   tongsocot = SmartTags("Blister_Show_Total_Blister_Column")	
   'tongsocot = 6
   '-------------------
   'bung = tongsocot - 1
   'If bung < 1 Then
   'bung = 1
   'End If
   '-------------------
   cycle = kc_hieudung / tongsocot '137
   Do_rong_cot = (cycle/3) *2		'91,3
   
   kc_2_cot = cycle		
   
   cot = tongsocot
   
   If tongsocot > 1 Then
   letrai = 50	
   Blis(tongsocot).width =  Do_rong_cot 
   	
   For i = 2  To tongsocot
   cot = cot - 1
   letrai = letrai + kc_2_cot
   
   Blis(cot).left =  letrai 
   Blis(cot).width = Do_rong_cot
   Next
   
   End If

VB script "Check_Lot"
   'Tip:
   ' 1. Use the <CTRL+SPACE> or <CTRL+I> shortcut to open a list of all objects and functions
   ' 2. Write the code using the HMI Runtime object.
   '  Example: HmiRuntime.Screens("Screen_1").
   ' 3. Use the <CTRL+J> shortcut to create an object reference.
   'Write the code as of this position:
   
   If SmartTags("Batch_Management_DB_Product_Name") <> "" And SmartTags("Batch_Management_DB_Batch_Number") <> "" And SmartTags("Batch_Management_DB_Lot_Size") > 0 Then
   SmartTags("Batch_Management_DB_B_Start_Lot") = True
   
   Else 
   SmartTags("Batch_Management_DB_B_Start_Lot") = False 
   bfde4b54-0db7-4817-8032-87127bf19bb9 "Chưa nhập đủ thông tin lô"
   End If

VB script "Write_Report"
   'Tip:
   ' 1. Use the <CTRL+SPACE> or <CTRL+I> shortcut to open a list of all objects and functions
   ' 2. Write the code using the HMI Runtime object.
   '  Example: HmiRuntime.Screens("Screen_1").
   ' 3. Use the <CTRL+J> shortcut to create an object reference.
   'Write the code as of this position:
    Const ForReading = 1, ForWriting = 2, ForAppending = 8
    Dim ngay, thang, nam, gio, phut, giay
    ngay = Day(Date)
    thang = Month(Date)
    nam = Year(Date)
    gio = Hour(Time)
    phut = Minute(Time)
    giay = Second(Time)
       Dim fs, f
       Set fs = CreateObject("Scripting.FileSystemObject")
       Set f = fs.OpenTextFile("E:\Test\abc.txt", ForAppending,True, -2)
       f.WriteLine CStr( CStr(ngay) + "/"+ CStr(thang) +"/"+ CStr(nam) + " "+ CStr(gio) + ":" + CStr(phut) +":" + CStr(giay))
       f.Close
*)